FUNCTION_BLOCK SampleComponentTests EXTENDS _internals_TcoContext
VAR
	_sut : TcoInspectors.SampleComponent(THIS^);
END_VAR

{attribute 'TcRpcEnable'}
METHOD INTERNAL AddTwoNumbersTest : INT
VAR_INPUT
	NumberOne : INT;
	NumberTwo : INT;
END_VAR
AddTwoNumbersTest := _sut.AddTwoNumbers(NumberOne, NumberTwo);
END_METHOD

METHOD PROTECTED Main
END_METHOD

{attribute 'TcRpcEnable'}
METHOD INTERNAL WaitForModuloTest : BOOL
VAR_INPUT
	Modulo : INT;
END_VAR
WaitForModuloTest := _sut.WaitForModulo(Modulo);
END_METHOD

END_FUNCTION_BLOCK

(* stored: Version 1.1.0.1, ProductVersion 3.1.4024.6
   POU SampleComponentTests: Id {8e88c5fb-6b37-0ee0-1dee-44bcdb0de8e4}, SpecialFunc None
   Method AddTwoNumbersTest: Id {e347ef7e-bfc9-0b26-39ae-1647a56bdbbd}
   Method Main: Id {2386eb08-ae25-07fa-0ae2-18bdce87e272}
   Method WaitForModuloTest: Id {a3e90fc3-609f-0e44-0b13-6aae397ca99c} *)
